(* PLC project Tc2_Utilities.INT64_TO_LREAL Demo, tc3-libraries-kb TwinCAT 3.1 *)
(* stored: creationDateTime 2026-05-10T17:00:00, modificationDateTime 2026-05-10T17:00:00 *)

PROGRAM P_Demo_INT64_TO_LREAL
  VAR
    rResult : LREAL;  (* INT64_TO_LREAL 返回值 *)
    bRun : BOOL;  (* 触发一次调用 *)
    ti : T_LARGE_INTEGER;  (* 测试用本地变量 *)
  END_VAR

            // ============================================================
// Tc2_Utilities.INT64_TO_LREAL 演示程序（FUNCTION）
// ============================================================
// 验证步骤：
//   1. 引用 Tc2_Utilities
//   2. 编译 + 登录
//   3. 强制 bRun := TRUE 一个周期
//   4. 在线监视 rResult
// ============================================================

ti := LARGE_INTEGER(0, 1234);
IF bRun THEN
    rResult := INT64_TO_LREAL(ti);
    bRun := FALSE;
END_IF;

          
END_PROGRAM
